TYPE DUT :
STRUCT
	cc:BOOL;
	dd:INT;
END_STRUCT
END_TYPE

(* stored: Version 1.1.0.1, ProductVersion 3.1.4024.6
   DUT DUT: Id {758145fa-aa88-4707-8007-b525cf0daefd} *)
